(* IEC 61131-3 sources: Industry-PLC-LLM/data/PLCBEAD_repo/PLCBEAD_PLCEmbed-main/PLC-BEAD/Source/GEB/GEN_PW2, 1 file *)

(* ---- GEN_PW2.ST ---- *)
FUNCTION UDINT_TO_TIME2:TIME

	VAR_INPUT
		IN :	UDINT;
	END_VAR

	UDINT_TO_TIME2 := DINT_TO_TIME(UDINT_TO_DINT(IN));

END_FUNCTION

FUNCTION_BLOCK T_PLC_MS_block
	VAR_OUTPUT
		T_PLC_MS :	UDINT;
	END_VAR

	VAR
		PLC_TICKS_PER_SEC :	INT;
		PLC_SYS_TICK_CNT :	DINT;
	END_VAR

	VAR
		debug :	BOOL;
		N :	INT;
		Offset :	UDINT;
		temp :	DWORD := DWORD#1;
		MODE :	BOOL;
		faktor :	UDINT;
		init :	BOOL;
		v_plc_ticks_per_sec :	UDINT;
		base :	UDINT := UDINT#1000;
	END_VAR

	IF init = FALSE THEN
		v_plc_ticks_per_sec := INT_TO_UDINT(PLC_TICKS_PER_SEC);
		IF v_plc_ticks_per_sec = UDINT#1024 THEN
			faktor := UDINT#1;
			MODE := FALSE;
		ELSIF v_plc_ticks_per_sec > UDINT#0 THEN
			IF v_plc_ticks_per_sec <= base THEN
				faktor := base / v_plc_ticks_per_sec;
				MODE := FALSE;
			ELSE
				faktor := v_plc_ticks_per_sec / base;
				MODE := TRUE;
			END_IF;
		ELSE
			faktor := UDINT#1;
		END_IF;
		init := TRUE;
	END_IF;

	IF MODE THEN
		T_PLC_MS := DINT_TO_UDINT(PLC_SYS_TICK_CNT) / faktor;
	ELSE
		T_PLC_MS := DINT_TO_UDINT(PLC_SYS_TICK_CNT) * faktor;
	END_IF;

	IF debug THEN
		T_PLC_MS := (DWORD_TO_UDINT(SHL(UDINT_TO_DWORD(T_PLC_MS),N) OR SHL(temp,N)) - UDINT#1) + Offset;
	END_IF;

END_FUNCTION_BLOCK

FUNCTION_BLOCK GEN_PW2_Block

	VAR_INPUT
		ENQ :	BOOL;
		TH1 :	TIME;
		TL1 :	TIME;
		TH2 :	TIME;
		TL2 :	TIME;
		TS :	BOOL;
	END_VAR

	VAR_OUTPUT
		Q :	BOOL;
		TH :	TIME;
		TL :	TIME;
	END_VAR

	VAR
		T_PLC_MS :	T_PLC_MS_block;
		t_HIGH :	TIME;
		t_LOW :	TIME;
		TX :	TIME;
		START :	TIME;
		init :	BOOL;
		et :	TIME;
	END_VAR

	T_PLC_MS();
	TX:= UDINT_TO_TIME(T_PLC_MS.T_PLC_MS);

	IF NOT init THEN
		START := TX;
		init := TRUE;
		TH := T#0s;
		TL := T#0s;
	END_IF;

	IF TS THEN
		t_HIGH := TH2;
		t_LOW := TL2;
	ELSE
		t_HIGH := TH1;
		t_LOW := TL1;
	END_IF;

	IF ENQ THEN
		et := SUB_TIME(TX , START);
		IF NOT Q THEN
			IF et >= t_LOW THEN
				Q := TRUE;
				START := TX;
				TL := T#0s;
			ELSE
				TL := et;
			END_IF;
		ELSE
			IF et >= t_HIGH THEN
				Q := FALSE;
				START := TX;
				TH := T#0s;
			ELSE
				TH := et;
			END_IF;
		END_IF;
	ELSE
		Q := FALSE;
		TH := T#0s;
		TL := T#0s;
		START := TX;
	END_IF;

END_FUNCTION_BLOCK

PROGRAM program0
  VAR
	ENQ :	BOOL;
	TH1 :	TIME;
	TL1 :	TIME;
	TH2 :	TIME;
	TL2 :	TIME;
	TS :	BOOL;
	Q :	BOOL;
	TH :	TIME;
	TL :	TIME;
	func_block : GEN_PW2_Block;
  END_VAR
	func_block.ENQ  :=ENQ;
	func_block.TH1  :=TH1;
	func_block.TL1  :=TL1;
	func_block.TH2  :=TH2;
	func_block.TL2  :=TL2;
	func_block.TS  :=TS;
	func_block.TS  :=TS;
	func_block();
	Q := func_block.Q;
	TH := func_block.TH;
	TL := func_block.TL;

END_PROGRAM
